// TIA Portal V20 export
DATA_BLOCK "OPCUA"   // DB900
TITLE = INTERFACE
{ S7_Optimized_Access := 'FALSE' }
AUTHOR : HYUNDAI-MOVEX
FAMILY : LGR
VERSION : 0.1
// stored: AutoNumber false, DBAccessibleFromOPCUA true, DBAccessibleFromWebserver false, IsOnlyStoredInLoadMemory false, IsWriteProtectedInAS false
   VAR
      GRM : Struct
         CMD : Struct
            NTP : "LGR_DTL";
            InterlockByGCS : Array[1..32] of "LGR_Interface_CV_PO";
         END_STRUCT;
         STAT : Struct
            NTP : DTL;
            CMDRetry : Array[1..3] of Bool;
            ForceUse : Array[1..2] of Bool;
            DoorOpened : Array[1..16] of Bool;
            StatusCode : "LGR_Equip_StatusDetail";
         END_STRUCT;
      END_STRUCT;
      GR : Array[1..3] of "LGR_Interface_GR";
      STATION : Array[1..32] of "LGR_STATION";
   END_VAR
BEGIN
END_DATA_BLOCK
